// Mitsubishi GX Works2 project: 1   PLC: Q02/Q02H

PROGRAM MAIN
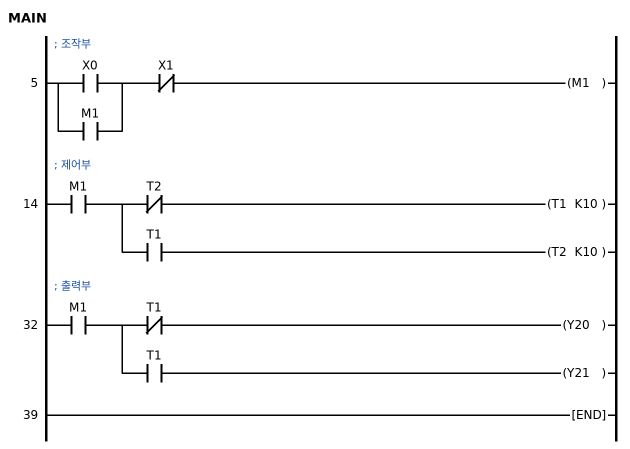
; 조작부
5     LD      X0
      OR      M1
      ANI     X1
      OUT     M1
; 제어부
14    LD      M1
      MPS
      ANI     T2
      OUT     T1 K10
      MPP
      AND     T1
      OUT     T2 K10
; 출력부
32    LD      M1
      MPS
      ANI     T1
      OUT     Y20
      MPP
      AND     T1
      OUT     Y21
39    END
END_PROGRAM
